// TIA Portal V19 export
DATA_BLOCK "PublishedDB"   // DB5
// stored: Access Published, MemoryReserve 100, Namespace Unit2
   VAR
      handlingXyzToNgConveyor { S7_SetPoint := 'True'} : "LEXCHANGETRAY_typeHandlingXyzEm_interface";
      rollerB1ToLogistic { S7_SetPoint := 'True'} : "LEXCHANGETRAY_typeRoller_interface";
      rollerB2ToLogistic { S7_SetPoint := 'True'} : "LEXCHANGETRAY_typeRoller_interface_B2";
   END_VAR
BEGIN
END_DATA_BLOCK
